TYPE sDatagridVFD :
STRUCT
	NameVFD 			: STRING;
	CurrentSpeed 		: INT;
	SpeedSetpointLow 	: INT;
	SpeedSetpointHigh 	: INT;
	
END_STRUCT
END_TYPE

(* stored: Version 1.1.0.1, ProductVersion 3.1.4024.12
   DUT sDatagridVFD: Id {82e68e44-fef3-4832-b2d2-c167662ab4e7} *)
